(* PLC project PLC411_SYS, home PLC411_SYS 1 *)
(* stored: creationDateTime 2023-04-11T08:18:12, productRelease 0, modificationDateTime 2023-04-11T08:26:49, version 1 *)

(* Программная перезагрузка устройства *)
FUNCTION SoftReset : BOOL
  VAR_INPUT
    Ex : BOOL := FALSE;  (* Разрешение исполнения *)
  END_VAR

            {extern void AppSys_SoftReset(BOOL);AppSys_SoftReset(EX);}
SoftReset:= TRUE;

          
END_FUNCTION

(* Управление LED_USER *)
FUNCTION_BLOCK LedUser
  VAR_INPUT
    V : BOOL := FALSE;  (* значение *)
  END_VAR
  VAR_OUTPUT
    Ov : BOOL := FALSE;  (* значение (установленное) *)
  END_VAR

            {extern void App_LedUser(LEDUSER*);App_LedUser(data__);}

          
END_FUNCTION_BLOCK
